# EPICS substitutions: apps/caenV65XXApp/Db/v6521.substitutions
file "db/v6521chan.db" {
pattern
 {CrName, Sl, Ch, high, hihi, low, lolo}
 {"HAHV95", "00", "000", "25", "50", "-50", "-25"}
 {"HAHV95", "00", "001", "25", "50", "-50", "-25"}
 {"HAHV95", "00", "002", "25", "50", "-50", "-25"}
 {"HAHV95", "00", "003", "25", "50", "-50", "-25"}
 {"HAHV95", "00", "004", "25", "50", "-50", "-25"}
 {"HAHV95", "00", "005", "25", "50", "-50", "-25"}
# {"HAHV95", "01", "000", "25", "50", "-50", "-25"}
# {"HAHV95", "01", "001", "25", "50", "-50", "-25"}
# {"HAHV95", "01", "002", "25", "50", "-50", "-25"}
# {"HAHV95", "01", "003", "25", "50", "-50", "-25"}
# {"HAHV95", "01", "004", "25", "50", "-50", "-25"}
# {"HAHV95", "01", "005", "25", "50", "-50", "-25"}
# {"HAHV95", "02", "000", "25", "50", "-50", "-25"}
# {"HAHV95", "02", "001", "25", "50", "-50", "-25"}
# {"HAHV95", "02", "002", "25", "50", "-50", "-25"}
# {"HAHV95", "02", "003", "25", "50", "-50", "-25"}
# {"HAHV95", "02", "004", "25", "50", "-50", "-25"}
# {"HAHV95", "02", "005", "25", "50", "-50", "-25"}
}
